Yaskawa INFORM job: R1_BATMAN_NOWY_KM-OK.JBI

/JOB
//NAME R1_BATMAN_NOWY_KM-OK
///FOLDERNAME KRIS-SCIANA
//POS
///NPOS 410,410,0,26,0,0
///TOOL 0
///POSTYPE PULSE
///PULSE
C00000=29960,139157,41546,-12188,94395,86333
C00001=12800,76505,-14321,-12731,99531,83391
C00002=-93330,-9337,26195,-7488,46800,71866
C00003=-109648,13515,16388,-582,84053,65182
C00004=-109670,16422,24252,-586,80707,65189
C00005=-109670,16934,25656,-587,80107,65191
C00006=-109670,16422,24252,-586,80707,65189
C00007=-110374,15664,24172,-576,80363,64950
C00008=-110374,13408,17598,-573,83249,64937
C00009=-100947,5020,18268,-732,78517,68109
C00010=-100947,5466,19407,-733,78046,68110
C00011=-100947,5020,18268,-732,78517,68109
C00012=-101669,3533,17505,-722,78217,67864
C00013=-100947,5020,18268,-732,78517,68109
C00014=-93324,28905,32784,-832,81932,70679
C00015=-94152,26793,37960,-831,77656,70427
C00016=-94152,27168,38874,-831,77287,70429
C00017=-94152,26793,37960,-831,77656,70427
C00018=-94428,25011,36465,-827,77656,70332
C00019=-94152,26793,37960,-831,77656,70427
C00020=-83677,18451,34531,-972,75597,74005
C00021=-83677,18852,35456,-973,75233,74007
C00022=-83677,18451,34531,-972,75597,74005
C00023=-84064,17163,33488,-967,75571,73871
C00024=-83677,18451,34531,-972,75597,74005
C00025=-81641,11244,27675,-995,76137,74695
C00026=-81493,11059,28179,-998,75733,74748
C00027=-81641,11244,27675,-995,76137,74695
C00028=-82191,12588,29665,-991,75598,74510
C00029=-81641,11244,27675,-995,76137,74695
C00030=-91711,-19484,9455,-889,71442,71303
C00031=-91372,-20164,10041,-896,70736,71423
C00032=-91711,-19484,9455,-889,71442,71303
C00033=-92389,-17223,12578,-883,70676,71076
C00034=-91711,-19484,9455,-889,71442,71303
C00035=-106821,23381,33578,-700,78719,66116
C00036=-140607,-14296,8355,17640,72856,-28938
C00037=-138803,-8748,20112,18029,68291,-28986
C00038=-139069,-9638,20936,18155,67425,-29218
C00039=-138803,-8748,20112,18029,68291,-28986
C00040=-138658,-6539,23170,18113,67548,-29051
C00041=-138803,-8748,20112,18029,68291,-28986
C00042=-151062,6621,28732,17951,73370,-32606
C00043=-147529,16835,48440,18711,66071,-32499
C00044=-147718,16293,48665,18768,65717,-32627
C00045=-147529,16835,48440,18711,66071,-32499
C00046=-147292,19253,51437,18794,65449,-32517
C00047=-147529,16835,48440,18711,66071,-32499
C00048=-160315,9548,45137,18676,67160,-36871
C00049=-160315,11416,48596,18832,66051,-37055
C00050=-160034,10639,48797,18917,65496,-37052
C00051=-160315,11416,48596,18832,66051,-37055
C00052=-159902,14249,52211,18957,65234,-37046
C00053=-160315,11416,48596,18832,66051,-37055
C00054=-160315,1266,28928,18053,72602,-36008
C00055=-155372,33863,69589,13242,72639,-71520
C00056=-155372,33877,69614,13243,72631,-71521
C00057=-155632,33114,69495,13228,72357,-71637
C00058=-155372,33877,69614,13243,72631,-71521
C00059=-154967,38534,75787,13400,71201,-71548
C00060=-155372,33877,69614,13243,72631,-71521
C00061=-155372,14771,31861,12741,85721,-70138
C00062=-144854,-16074,11616,14078,80727,-67113
C00063=-144738,-11911,19372,14194,78150,-67371
C00064=-144388,-8955,22802,14262,77515,-67327
C00065=-144738,-11911,19372,14194,78150,-67371
C00066=-145031,-12965,19294,14184,77720,-67519
C00067=-144738,-11911,19372,14194,78150,-67371
C00068=-144738,-22241,-3507,13967,86670,-66398
C00069=-137755,-5473,21324,14836,78997,-64910
C00070=-137072,-7723,19533,14904,78825,-64700
C00071=-137755,-5473,21324,14836,78997,-64910
C00072=-137755,-4185,24016,14880,78032,-65028
C00073=-137755,-5473,21324,14836,78997,-64910
C00074=-136397,694,15927,14772,85041,-63716
C00075=-136397,302,14935,14766,85437,-63669
C00076=-109887,-1557,13389,16194,80395,55204
C00077=-88793,-1230,14928,-10868,86441,64286
C00078=-87997,13509,39457,-13767,84419,65011
C00079=-88765,12150,38219,-13907,84356,64763
C00080=-87997,13509,39457,-13767,84419,65011
C00081=-87997,14649,41772,-13784,83604,65104
C00082=-87997,13509,39457,-13767,84419,65011
C00083=-87997,4090,18260,-13774,92399,64126
C00084=-90135,-15090,27302,-19288,66922,75027
C00085=-93339,-8581,40987,-20291,61446,74887
C00086=-93414,13551,61682,-18148,70133,73308
C00087=-93501,10236,57492,-18075,70950,73153
C00088=-74509,-9574,47474,-19286,61435,81215
C00089=-71490,563,57958,-19102,60836,82318
C00090=-73930,26348,84328,-20021,57559,82128
C00091=-53296,23546,81196,-16554,61634,87978
C00092=-53399,1993,45500,-15348,72112,86487
C00093=-93772,6441,51176,-23543,71504,29074
C00094=-93782,7493,53021,-23621,70954,29184
C00095=-97809,11823,34750,-18310,96930,22381
C00096=-97765,18036,47284,-18125,92636,23039
C00097=-93436,10227,57510,-23741,69792,29543
C00098=-92885,10092,58329,-23719,69400,29810
C00099=-94577,32380,63989,-17035,90534,24406
C00100=-93990,31397,63393,-16840,90513,24603
C00101=-86403,12665,47397,-14267,92055,26863
C00102=-83940,7836,43519,-13404,92349,27621
C00103=-88022,26657,64193,-8590,95838,24607
C00104=-86621,7360,57775,-7913,90052,25407
C00105=-86874,-9205,28605,-8179,99382,24730
C00106=-93784,11972,60674,-23958,68741,29649
C00107=-120720,1752,25513,-527,80353,-9094
C00108=-141476,7352,24714,17219,80156,-38332
C00109=-140652,10872,31760,17392,77568,-38413
C00110=-151911,2048,28558,16772,77396,-42350
C00111=-153373,1194,28316,16661,77408,-42852
C00112=-154278,885,28252,16586,77468,-43151
C00113=-151033,405,27146,8511,73769,-41301
C00114=-151062,615,27322,8509,73772,-41310
C00115=-152803,25350,52147,11197,72163,-42431
C00116=-157202,33761,63402,16632,73491,-44702
C00117=-172575,32003,68245,15007,72491,-49961
C00118=-172661,17404,41016,14506,81470,-48897
C00119=-145328,-17018,3942,17006,81208,-68726
C00120=-143820,-16511,8308,17205,78576,-68574
C00121=-147802,-4731,19998,17005,78294,-69996
C00122=-143624,-15596,9649,11345,73102,-68510
C00123=-152471,-38163,-4132,7931,70088,-70764
C00124=-152752,-37985,-4023,7933,70138,-70858
C00125=-161611,-21890,10565,15904,78087,-74768
C00126=-170415,38593,75058,15377,71350,-78588
C00127=-170289,22176,44233,14795,81516,-77278
C00128=-170289,11960,19922,14705,90922,-76157
C00129=16919,130033,39084,-10517,94456,75601
C00130=16919,130033,39084,-10517,94456,75601
C00131=-97369,-13902,24194,28978,70576,-6709
C00132=-95632,-2500,42487,30176,65295,-7505
C00133=-95207,2788,47639,30323,64767,-7497
C00134=-94456,3304,48081,30401,64521,-7286
C00135=-95207,2788,47639,30323,64767,-7497
C00136=-94939,4605,50640,30565,63888,-7653
C00137=-95207,2788,47639,30323,64767,-7497
C00138=-103162,11339,55190,29411,67038,-9800
C00139=-102527,20996,70482,30499,62962,-10725
C00140=-102527,23747,75000,30853,61778,-11081
C00141=-102527,20996,70482,30499,62962,-10725
C00142=-101170,23554,74068,30934,61779,-10587
C00143=-102527,20996,70482,30499,62962,-10725
C00144=-108080,-3135,57545,30673,60740,-13355
C00145=-107519,-2528,59016,30963,60068,-13361
C00146=-108080,-3135,57545,30673,60740,-13355
C00147=-108548,-1030,60547,30798,60211,-13680
C00148=-108080,-3135,57545,30673,60740,-13355
C00149=-118454,-19329,55183,30459,57655,-17824
C00150=-117324,-18814,56509,30922,56888,-17699
C00151=-118454,-19329,55183,30459,57655,-17824
C00152=-118779,-17072,58124,30582,57172,-18080
C00153=-118454,-19329,55183,30459,57655,-17824
C00154=-119568,-37031,32608,28877,62130,-16877
C00155=-139069,-33471,54850,26577,56126,-24455
C00156=-140948,-25344,66415,26849,53845,-25589
C00157=-140947,-22345,70767,27227,52824,-25875
C00158=-140948,-25344,66415,26849,53845,-25589
C00159=-138778,-24772,68372,27918,52625,-25364
C00160=-140948,-28933,61200,26421,55072,-25252
C00161=-139172,-36190,52504,26531,56189,-82791
C00162=-107699,-48855,44139,22027,38536,-72276
C00163=-109632,-48276,45968,22227,38076,-73074
C00164=-107699,-48855,44139,22027,38536,-72276
C00165=-107022,-47413,45796,22221,38170,-72148
C00166=-107699,-48855,44139,22027,38536,-72276
C00167=-87180,-57379,25744,20107,41611,-64125
C00168=-87177,-56321,27969,20431,40831,-64319
C00169=-87180,-57379,25744,20107,41611,-64125
C00170=-86636,-54726,28428,20224,41246,-64016
C00171=-87180,-57379,25744,20107,41611,-64125
C00172=-68556,-59148,10398,16762,46593,-56068
C00173=-68720,-58452,12286,16994,45847,-56271
C00174=-68556,-59148,10398,16762,46593,-56068
C00175=-67991,-57295,12403,16799,46232,-55922
C00176=-68556,-59148,10398,16762,46593,-56068
C00177=-65065,-64227,-6791,14726,53714,-53588
C00178=-61076,-57425,2885,14865,50705,-52539
C00179=-61164,-57495,4364,15074,49802,-52712
C00180=-61076,-57425,2885,14865,50705,-52539
C00181=-60686,-55325,4818,14851,50535,-52416
C00182=-61076,-57425,2885,14865,50705,-52539
C00183=-61076,-73603,-22996,13552,58097,-51511
C00184=-82396,-73217,-22842,14872,61637,60164
C00185=-87516,-60977,-6284,80955,41162,78434
C00186=-74092,-52490,8277,91201,32262,75613
C00187=-78785,-42356,17001,89628,35140,75415
C00188=-77330,-41476,17474,89941,34254,75571
C00189=-78785,-42356,17001,89628,35140,75415
C00190=-78785,-39715,21246,91443,35108,74420
C00191=-78785,-42356,17001,89628,35140,75415
C00192=-88814,-14584,37421,84097,41483,76258
C00193=-87600,-13774,38015,84402,40735,76362
C00194=-88814,-14584,37421,84097,41483,76258
C00195=-88814,-11485,42642,85948,41288,75148
C00196=-88814,-14584,37421,84097,41483,76258
C00197=-88814,-12912,40245,85098,41370,75657
C00198=-87720,-12181,40790,85402,40703,75739
C00199=-88814,-12912,40245,85098,41370,75657
C00200=-88814,-10194,44789,86704,41222,74694
C00201=-88814,-12912,40245,85098,41370,75657
C00202=-81268,8239,25602,62836,54247,42871
C00203=-99383,-12682,5103,58765,66557,41036
C00204=-74635,2773,19953,61588,50422,44547
C00205=-74870,7103,29898,71541,48579,40569
C00206=-73722,4389,21160,61383,49897,44786
C00207=-73275,4966,21408,61205,49691,44957
C00208=-83489,55985,81914,76438,52196,35596
C00209=-80400,36125,52423,64197,52680,41941
C00210=-80398,36126,52424,64197,52679,41941
C00211=-78951,-40444,4950,38310,62421,-17800
C00212=-78960,-34903,14668,39360,59955,-18811
C00213=-72845,-10333,24086,24565,76568,-49529
C00214=-69730,1194,40732,25450,71769,-49472
C00215=-79919,-36306,13442,39288,60368,-19058
C00216=-79943,-36084,12678,39084,60835,-18874
C00217=-86153,35123,85647,24141,66737,-56179
C00218=-71006,-12268,19845,19209,73235,-48605
C00219=-78486,-5699,27880,17849,72527,-51167
C00220=-84137,3114,38840,17597,71558,-53260
C00221=-84122,-12372,4412,16852,84221,-51450
C00222=-94700,16963,33528,63705,62536,40249
C00223=-80389,36149,52448,64198,52673,41941
C00224=-80398,36126,52424,64197,52679,41941
C00225=-82543,39244,62629,76344,52787,36963
C00226=-83474,48309,76175,82007,53048,34101
C00227=-80829,34452,49584,63632,53361,42311
C00228=-80419,35008,49905,63542,53144,42433
C00229=-83495,46424,73588,81542,53170,34449
C00230=-83461,45298,72093,81297,53209,34643
C00231=-83534,45148,71928,81265,53263,34652
C00232=-83974,39234,63618,79687,53967,35775
C00233=-87946,20987,32632,62140,59518,42667
C00234=-98278,19923,28034,11913,78019,-9874
C00235=-92244,58536,75756,7832,70371,-3504
C00236=-91977,78904,104422,8238,63238,-3903
C00237=-107781,18098,54792,50122,40570,-59241
C00238=-108140,20187,57804,50894,40242,-59767
C00239=-92594,57126,80356,8020,66880,-3859
C00240=-94908,21990,48768,7976,68471,-4548
C00241=-98306,-6406,30616,8206,65402,-5929
C00242=-103070,-28468,23138,8725,59186,-8038
C00243=-105710,-35465,21971,8985,56591,-9160
C00244=-105525,-39817,14322,8753,59014,-8895
C00245=-105525,-70728,-42035,7727,77630,-7598
C00246=-78386,25843,42020,64423,60972,44329
C00247=-85759,14880,31595,64053,66010,43452
C00248=-85595,16938,42729,82497,65241,37214
C00249=-81136,28617,59931,85714,61589,35095
C00250=-78173,23730,38609,63927,61301,44837
C00251=-78597,23175,38323,63988,61519,44714
C00252=-72881,-4192,29043,86400,56225,36548
C00253=-67760,-16410,19348,87784,52710,36541
C00254=-59662,-27119,-2583,63857,48640,46851
C00255=-59488,-28058,-2749,64137,48352,46679
C00256=-60158,-29069,10200,71536,45362,41690
C00257=-61387,-28761,11042,71804,46022,41293
C00258=-67092,-34207,-766,67938,51323,42934
C00259=-57818,-28976,-3296,38246,61056,30495
C00260=-70399,-33004,-19929,37727,73042,29338
C00261=-119023,5793,43031,54634,61324,54134
C00262=-110425,23913,49460,37198,87531,-1667
C00263=-103784,36935,71027,39124,79569,-1855
C00264=-107895,22032,60540,56797,53926,55382
C00265=-107775,18111,54805,55911,54728,56108
C00266=-104144,33311,68301,39058,79572,-1995
C00267=-105177,26013,62623,38825,79784,-2330
C00268=-105381,26208,63001,38785,79763,-2415
C00269=-106285,20699,59223,38608,79730,-2777
C00270=-106624,19858,58731,38534,79764,-2897
C00271=-106746,20912,59987,38524,79628,-2990
C00272=-106325,7794,45978,38293,75046,-4276
C00273=-104338,-11348,28641,37974,64498,-6611
C00274=-104860,-11037,29608,38068,64365,-6884
C00275=-107519,-11058,32205,38335,64151,-8093
C00276=-107851,-11129,32812,38426,63958,-8307
C00277=-116434,-38739,5593,36913,69412,-9812
C00278=-124683,-63657,-10921,36340,70465,-12735
C00279=-150183,-86751,-58871,11994,78291,3293
C00280=-2356,-86751,-58871,11994,78291,3293
C00281=12334,49205,1562,-2559,87983,53268
C00282=-150183,-86751,-58871,11994,78291,3293
C00283=-131366,13830,22994,-19726,75607,38471
C00284=-136534,55496,89709,-36696,55641,43467
C00285=-137035,56054,90375,-36738,55351,43362
C00286=-136534,55496,89709,-36696,55641,43467
C00287=-136534,59618,96436,-37542,54010,44136
C00288=-136534,55496,89709,-36696,55641,43467
C00289=-145752,56924,83291,-5552,58900,12813
C00290=-147360,56365,85008,-5446,57459,12300
C00291=-147195,60965,91580,-5568,55798,12447
C00292=-147360,56365,85008,-5446,57459,12300
C00293=-147752,57421,87154,-5449,56660,12196
C00294=-147360,56365,85008,-5446,57459,12300
C00295=-144876,20699,52980,-5661,58991,13126
C00296=-144465,22925,56598,-5771,57941,13331
C00297=-144876,20699,52980,-5661,58991,13126
C00298=-145346,20760,54373,-5658,58141,13001
C00299=-144876,20699,52980,-5661,58991,13126
C00300=-140458,-9363,35089,-6525,54898,15024
C00301=-139844,-7295,37930,-6647,54260,15291
C00302=-140458,-9363,35089,-6525,54898,15024
C00303=-141162,-9224,36313,-6501,54169,14811
C00304=-140458,-9363,35089,-6525,54898,15024
C00305=-124022,-11653,42832,-20763,58582,23587
C00306=-123999,-9443,45795,-20909,57941,23722
C00307=-124022,-11653,42832,-20763,58582,23587
C00308=-124750,-10986,44233,-20923,57940,23461
C00309=-124022,-11653,42832,-20763,58582,23587
C00310=-120425,-27436,23026,-19779,63062,73790
C00311=-124426,-21462,36323,-21031,57405,73472
C00312=-124464,-21490,37251,-21166,56849,73573
C00313=-124426,-21462,36323,-21031,57405,73472
C00314=-125014,-20092,38108,-21159,56911,73366
C00315=-124426,-21462,36323,-21031,57405,73472
C00316=-142818,-53721,4956,-21021,55965,67145
C00317=-142626,-53506,6347,-21202,55310,67354
C00318=-142818,-53721,4956,-21021,55965,67145
C00319=-143779,-52181,6747,-21095,55463,66895
C00320=-142818,-53721,4956,-21021,55965,67145
C00321=-174971,-75680,-15206,-18859,50174,56027
C00322=-175130,-75408,-13794,-19036,49449,56108
C00323=-174971,-75680,-15206,-18859,50174,56027
C00324=-175277,-74010,-13504,-18872,49932,55952
C00325=-174971,-75680,-15206,-18859,50174,56027
C00326=-173245,-86721,-27893,-18523,52547,56249
C00327=-203888,-83968,-26454,-13077,47682,44754
C00328=-205019,-83483,-25221,-12917,47022,44380
C00329=-203888,-83968,-26454,-13077,47682,44754
C00330=-204234,-82255,-25110,-12985,47684,44611
C00331=-203888,-83968,-26454,-13077,47682,44754
C00332=-178857,-84729,-36876,-16471,57715,53184
C00333=-172192,-78951,-17187,-49367,43626,66497
C00334=-173896,-78013,-16876,-49026,43021,65876
C00335=-172192,-78951,-17187,-49367,43626,66497
C00336=-172192,-77329,-14763,-49894,43190,66824
C00337=-172192,-78951,-17187,-49367,43626,66497
C00338=-162487,-85150,-21286,-50022,47755,69383
C00339=-141360,-58545,-9704,-51911,39719,82506
C00340=-155475,-48260,1081,-49396,31731,78582
C00341=-156810,-47533,1467,-48693,31169,77981
C00342=-155475,-48260,1081,-49396,31731,78582
C00343=-155475,-46586,3939,-50523,31140,79172
C00344=-155475,-48260,1081,-49396,31731,78582
C00345=-143506,-57069,-7972,-51767,38422,82026
C00346=-132998,-15066,34811,-73278,45446,90463
C00347=-136647,7793,53326,-73557,43352,89771
C00348=-137414,8138,53635,-73690,42883,89678
C00349=-136647,7793,53326,-73557,43352,89771
C00350=-136647,9971,57074,-74779,42995,90526
C00351=-136647,7793,53326,-73557,43352,89771
C00352=-127315,-7809,27658,-65953,51971,86730
C00353=-123754,-52231,-17316,-40750,89865,-5838
C00354=-130215,-25533,26580,-55595,80666,-780
C00355=-127399,30151,75869,-54823,81081,357
C00356=-123761,23089,64182,-53294,85068,-318
C00357=-107579,-13362,25214,-39024,97613,11163
C00358=-170043,-71406,-31414,-11284,81739,48155
C00359=-190061,-61831,-15348,-14174,73926,42337
C00360=-162764,-46045,3348,-10421,74427,51168
C00361=-141001,-25000,21572,-6477,76090,57905
C00362=-128005,1092,47071,-3936,74564,61986
C00363=-123328,16053,63213,-3007,72497,63466
C00364=-123444,-5699,22378,-2915,86428,63100
C00365=-123444,-16678,-3411,-2947,96644,62863
C00366=-133517,-66572,-32265,-38878,44642,78881
C00367=-132900,-49128,-445,-67646,40881,87931
C00368=-134943,-41043,7919,-68788,39256,88202
C00369=-129486,24309,60482,-67313,43043,88408
C00370=-129295,28550,64902,-67843,42938,88773
C00371=-124005,7439,40047,-63776,48062,87191
C00372=-119115,-2939,24898,-61013,52949,86096
C00373=-132234,15475,18840,-9177,73687,21564
C00374=-138193,54177,73040,-9110,59720,20493
C00375=-142429,56695,78528,-2248,54886,15330
C00376=-135428,11470,41007,-7421,55168,18590
C00377=-124358,-15323,27893,-15893,51961,24324
C00378=-114489,-24173,28344,-21843,50628,29378
C00379=-104693,-29158,30498,-25923,50747,33967
C00380=-104394,-36428,19495,-24933,53579,33323
C00381=-104394,-63765,-28743,-21562,68022,30158
C00382=-137801,-54017,-22800,-32811,77180,42551
C00383=-145098,-49977,-15343,-33510,72300,41124
C00384=-157536,-82053,-30611,-35478,61676,39542
C00385=-167332,-94403,-34954,-36782,54951,37849
C00386=-168775,-95552,-35063,-36976,53981,37598
C00387=-175265,-101786,-36159,-35767,45251,37123
C00388=-172094,-106020,-33228,-38547,43201,39696
C00389=-170782,-105999,-32632,-38876,43404,40255
C00390=-154100,-109404,-39309,-37897,51447,44344
C00391=-127200,-116118,-56301,-33842,67042,49701
C00392=-160521,-112920,-64126,-13181,65496,7682
C00393=-193283,-91966,-46197,-10210,60672,-3708
C00394=-179428,-87326,-33956,-22991,51575,4568
C00395=-182309,-93219,-32914,-23693,47463,4374
C00396=-181968,-93619,-32743,-23870,47264,4575
C00397=-184128,-96951,-32374,-24207,44941,4267
C00398=-184601,-97825,-32091,-24365,44249,4253
C00399=-192271,-94092,-34086,-15205,49403,-1377
C00400=-156461,-94996,-22149,-46235,47288,20425
C00401=-143339,-75495,-15964,-42086,57329,21373
C00402=-155681,-87382,-19579,-43513,38484,12104
C00403=-154383,-87178,-18470,-44197,38599,12813
C00404=-148677,-87335,-15888,-46202,39785,15423
C00405=-143679,-101658,-25353,-47688,40824,17641
C00406=-91918,-122697,-50228,-39868,65277,29334
C00407=-93784,-22748,-9129,-22507,91967,25137
C00408=5840,107598,31668,-14199,93922,74405
C00409=29960,139157,41546,-12188,94395,86333
BC00000=68533,13783,1075157
BC00001=137001,15545,1050957
BC00002=200108,21911,920879
BC00003=200107,21911,776849
BC00004=200107,21911,776849
BC00005=200107,21911,776849
BC00006=200107,21911,776849
BC00007=200107,21911,776849
BC00008=200107,21911,776849
BC00009=199824,21894,777489
BC00010=199824,21894,777489
BC00011=199824,21894,777489
BC00012=199824,21894,777489
BC00013=199824,21894,777489
BC00014=199824,21894,743092
BC00015=199824,21894,743092
BC00016=199824,21894,743092
BC00017=199824,21894,743092
BC00018=199824,21894,743092
BC00019=199824,21894,743092
BC00020=199824,21894,743092
BC00021=199824,21894,743092
BC00022=199824,21894,743092
BC00023=199824,21894,743092
BC00024=199824,21894,743092
BC00025=199824,21894,743092
BC00026=199824,21894,743092
BC00027=199824,21894,743092
BC00028=199824,21894,743092
BC00029=199824,21894,743092
BC00030=199824,21894,835261
BC00031=199824,21894,835261
BC00032=199824,21894,835261
BC00033=199824,21894,835261
BC00034=199824,21894,835261
BC00035=199824,21894,835261
BC00036=199824,21894,835261
BC00037=199824,21894,835261
BC00038=199824,21894,835261
BC00039=199824,21894,835261
BC00040=199824,21894,835261
BC00041=199824,21894,835261
BC00042=199824,21894,835261
BC00043=199824,21894,835261
BC00044=199824,21894,835261
BC00045=199824,21894,835261
BC00046=199824,21894,835261
BC00047=199824,21894,835261
BC00048=199824,21894,835261
BC00049=199824,21894,835261
BC00050=199824,21894,835261
BC00051=199824,21894,835261
BC00052=199824,21894,835261
BC00053=199824,21894,835261
BC00054=199824,21894,835261
BC00055=199824,21894,835261
BC00056=199824,21894,835261
BC00057=199824,21894,835261
BC00058=199824,21894,835261
BC00059=199824,21894,835261
BC00060=199824,21894,835261
BC00061=199824,21894,835261
BC00062=199824,21894,835261
BC00063=199824,21894,835261
BC00064=199824,21894,835261
BC00065=199824,21894,835261
BC00066=199824,21894,835261
BC00067=199824,21894,835261
BC00068=199824,21894,835261
BC00069=199824,21895,835258
BC00070=199824,21895,835258
BC00071=199824,21895,835258
BC00072=199824,21895,835258
BC00073=199824,21895,835258
BC00074=199824,21895,835258
BC00075=199824,21895,835258
BC00076=199824,21895,835258
BC00077=199824,21895,835258
BC00078=199824,21895,835258
BC00079=199824,21895,835258
BC00080=199824,21895,835258
BC00081=199824,21895,835258
BC00082=199824,21895,835258
BC00083=199824,21895,835258
BC00084=205692,85135,967220
BC00085=205692,85135,967220
BC00086=205692,85135,967220
BC00087=205692,85135,967220
BC00088=205902,84947,966975
BC00089=205902,84947,966975
BC00090=205902,84947,966975
BC00091=205901,84948,926900
BC00092=205901,84948,926900
BC00093=218485,27554,1075175
BC00094=218485,27554,989857
BC00095=212076,30602,851577
BC00096=212076,30602,851577
BC00097=212075,30604,960971
BC00098=212075,30604,960971
BC00099=212076,30603,851574
BC00100=212076,30603,851574
BC00101=212076,30603,851572
BC00102=212076,30603,851571
BC00103=212076,30603,851571
BC00104=269506,91403,851571
BC00105=269506,91403,851571
BC00106=228143,33934,978152
BC00107=228143,33934,890863
BC00108=228143,33934,823600
BC00109=228143,33934,823600
BC00110=228143,33934,823600
BC00111=228143,33934,823600
BC00112=228143,33934,823600
BC00113=228143,33934,823600
BC00114=228143,33934,823600
BC00115=228144,33934,823598
BC00116=228144,33934,823598
BC00117=228144,33934,823598
BC00118=228144,33934,823598
BC00119=228144,33934,823598
BC00120=228144,33934,823598
BC00121=228144,33934,823598
BC00122=228144,33934,823598
BC00123=228144,33934,823598
BC00124=228144,33934,823598
BC00125=228144,33934,823598
BC00126=228144,33934,823598
BC00127=228144,33934,823598
BC00128=228144,33934,918948
BC00129=81693,35088,1064811
BC00130=81693,35088,1064811
BC00131=268670,144197,1015710
BC00132=268670,144197,1015710
BC00133=268670,144197,1015710
BC00134=268670,144197,1015710
BC00135=268670,144197,1015710
BC00136=268670,144197,1015710
BC00137=268670,144197,1015710
BC00138=268670,144196,1015709
BC00139=268670,144196,1015709
BC00140=268670,144196,1015709
BC00141=268670,144196,1015709
BC00142=268670,144196,1015709
BC00143=268670,144196,1015709
BC00144=268670,144196,1015709
BC00145=268669,144195,1015708
BC00146=268670,144196,1015709
BC00147=268670,144196,1015709
BC00148=268670,144196,1015709
BC00149=268670,144196,1015709
BC00150=268670,144196,1015709
BC00151=268670,144196,1015709
BC00152=268670,144196,1015709
BC00153=268670,144196,1015709
BC00154=268670,144196,1015709
BC00155=268670,144196,1015709
BC00156=268670,144196,1015709
BC00157=268670,144196,1015708
BC00158=268670,144196,1015709
BC00159=268670,144196,1015709
BC00160=268670,144196,1015709
BC00161=268670,144196,1015709
BC00162=268670,144196,1015709
BC00163=268670,144196,1015709
BC00164=268670,144196,1015709
BC00165=268670,144196,1015709
BC00166=268670,144196,1015709
BC00167=268669,113243,1015707
BC00168=268669,113243,1015707
BC00169=268669,113243,1015707
BC00170=268669,113243,1015707
BC00171=268669,113243,1015707
BC00172=268670,72970,1015708
BC00173=268670,72970,1015708
BC00174=268670,72970,1015708
BC00175=268670,72970,1015708
BC00176=268670,72970,1015708
BC00177=268670,48316,1015709
BC00178=268670,48316,1015709
BC00179=268670,48316,1015709
BC00180=268670,48316,1015709
BC00181=268670,48316,1015709
BC00182=268670,48316,1015709
BC00183=268670,48316,1015709
BC00184=268670,48316,1015709
BC00185=220078,15,922795
BC00186=227337,15,912089
BC00187=230240,15,907806
BC00188=230240,15,907806
BC00189=230240,15,907806
BC00190=230240,15,907806
BC00191=230240,15,907806
BC00192=230240,50273,907806
BC00193=230240,50273,907806
BC00194=230240,50273,907806
BC00195=230240,50273,907806
BC00196=230240,50273,907806
BC00197=230240,113905,907806
BC00198=230240,113905,907806
BC00199=230240,113905,907806
BC00200=230240,113905,907806
BC00201=230240,113905,907806
BC00202=173944,15,921053
BC00203=173944,15,921053
BC00204=178824,15,792329
BC00205=180775,15,783854
BC00206=180775,15,783854
BC00207=180775,15,783854
BC00208=180775,20545,783854
BC00209=179033,31181,784483
BC00210=174154,30731,805671
BC00211=235405,15,1075175
BC00212=235405,15,1001205
BC00213=235405,15,1001205
BC00214=235405,15,1001205
BC00215=243821,15,976624
BC00216=243821,15,976624
BC00217=235405,15,1001205
BC00218=196817,56536,842735
BC00219=189615,67087,813156
BC00220=189615,67087,813156
BC00221=189615,67087,813156
BC00222=174140,26317,913732
BC00223=174140,26317,913732
BC00224=174140,26317,806198
BC00225=179019,26768,785009
BC00226=180971,26948,776534
BC00227=180971,26948,776534
BC00228=180971,26948,776534
BC00229=181150,62034,771629
BC00230=181286,88704,767900
BC00231=181286,91968,766556
BC00232=177104,86088,775373
BC00233=174349,92139,798351
BC00234=257727,78000,903004
BC00235=258272,77360,890255
BC00236=258272,77360,890255
BC00237=262417,85815,884854
BC00238=262417,85815,884854
BC00239=258272,77360,890254
BC00240=258271,77360,890253
BC00241=258271,77360,890253
BC00242=258271,77360,890253
BC00243=258271,77360,890253
BC00244=258271,77360,890253
BC00245=258271,77360,890253
BC00246=174013,15,918199
BC00247=174013,15,810664
BC00248=180838,15,781222
BC00249=180838,15,781222
BC00250=180838,15,781222
BC00251=180838,15,781222
BC00252=180838,15,781222
BC00253=180838,15,781222
BC00254=180838,15,781222
BC00255=180838,15,781222
BC00256=180838,15,836511
BC00257=180838,15,836511
BC00258=180838,15,836511
BC00259=197117,15,902644
BC00260=197118,16,902641
BC00261=268113,94143,1075175
BC00262=276934,120699,948945
BC00263=276934,120699,948945
BC00264=274036,93127,945393
BC00265=274036,93127,945393
BC00266=276934,120699,948945
BC00267=276934,120699,948945
BC00268=276934,120699,948945
BC00269=276934,120699,948945
BC00270=276934,120699,948945
BC00271=276934,120699,948945
BC00272=276967,133711,947374
BC00273=277023,156083,944672
BC00274=277023,156083,944672
BC00275=277023,156083,944672
BC00276=277023,156083,944672
BC00277=277023,156083,944672
BC00278=277023,156083,944672
BC00279=277023,156083,944672
BC00280=135439,156083,1063650
BC00281=51795,156431,1068049
BC00282=277023,156083,944672
BC00283=173944,70115,921053
BC00284=173945,70115,925166
BC00285=173945,70115,925166
BC00286=173945,70115,925166
BC00287=173945,70115,925166
BC00288=173945,70115,925166
BC00289=173945,70115,921050
BC00290=173945,70115,921050
BC00291=173945,70115,921050
BC00292=173945,70115,921050
BC00293=173945,70115,921050
BC00294=173945,70115,921050
BC00295=173945,70115,921050
BC00296=173945,70115,921050
BC00297=173945,70115,921050
BC00298=173945,70115,921050
BC00299=173945,70115,921050
BC00300=173945,70115,921050
BC00301=173945,70115,921050
BC00302=173945,70115,921050
BC00303=173945,70115,921050
BC00304=173945,70115,921050
BC00305=173945,70115,921050
BC00306=173945,70115,921050
BC00307=173945,70115,921050
BC00308=173945,70115,921050
BC00309=173945,70115,921050
BC00310=173945,70115,921050
BC00311=173945,70115,921050
BC00312=173945,70115,921050
BC00313=173945,70115,921050
BC00314=173945,70115,921050
BC00315=173945,70115,921050
BC00316=173945,70115,921050
BC00317=173945,70115,921050
BC00318=173945,70115,921050
BC00319=173945,70115,921050
BC00320=173945,70115,921050
BC00321=173945,70115,921050
BC00322=173945,70115,921050
BC00323=173945,70115,921050
BC00324=173945,70115,921050
BC00325=173945,70115,921050
BC00326=173945,70115,921050
BC00327=173946,70115,921047
BC00328=173946,70115,921047
BC00329=173946,70115,921047
BC00330=173946,70115,921047
BC00331=173946,70115,921047
BC00332=173945,70114,921040
BC00333=173945,70114,921040
BC00334=173945,70114,921040
BC00335=173945,70114,921040
BC00336=173945,70114,921040
BC00337=173945,70114,921040
BC00338=173945,70114,921040
BC00339=173945,70114,921040
BC00340=173945,70114,921040
BC00341=173945,70114,921040
BC00342=173945,70114,921040
BC00343=173945,70114,921040
BC00344=173945,70114,921040
BC00345=173945,70114,921040
BC00346=173945,70114,921040
BC00347=173945,70114,921040
BC00348=173945,70114,921040
BC00349=173945,70114,921040
BC00350=173945,70114,921040
BC00351=173945,70114,921040
BC00352=173945,70114,921040
BC00353=153115,57298,944672
BC00354=153115,57298,944672
BC00355=153115,57298,944672
BC00356=153115,57298,944672
BC00357=153115,57298,944672
BC00358=153115,57298,944672
BC00359=153116,57298,944671
BC00360=153116,57298,944671
BC00361=153116,57298,916437
BC00362=153116,57298,892257
BC00363=153116,57298,881120
BC00364=153116,57298,881120
BC00365=153116,57298,881120
BC00366=153116,57298,881120
BC00367=153116,57298,881120
BC00368=153116,57298,881120
BC00369=153116,57298,881120
BC00370=153116,57298,881120
BC00371=153116,57298,881120
BC00372=153116,57298,881120
BC00373=153116,57298,881120
BC00374=153116,57298,881120
BC00375=153116,57298,881120
BC00376=153116,57299,881116
BC00377=153116,57299,881118
BC00378=153116,57298,881119
BC00379=153116,57298,881120
BC00380=153116,57298,881120
BC00381=153116,57298,881120
BC00382=153116,57298,881120
BC00383=153116,57298,881120
BC00384=153116,57298,881120
BC00385=153116,57298,881120
BC00386=153116,57298,881120
BC00387=153116,57298,881120
BC00388=153116,57298,881120
BC00389=153116,57298,881120
BC00390=153116,57298,881120
BC00391=153116,57298,881120
BC00392=155122,228922,881120
BC00393=155122,228922,881120
BC00394=155122,228922,881120
BC00395=155122,228922,881120
BC00396=155122,228922,881120
BC00397=155122,228922,881120
BC00398=155122,228922,881120
BC00399=155122,228922,881120
BC00400=155121,228922,881118
BC00401=155121,228922,881118
BC00402=155121,228922,881118
BC00403=155121,228922,881118
BC00404=155121,228922,881118
BC00405=155121,228922,881118
BC00406=155107,227689,881118
BC00407=228143,33934,978152
BC00408=99644,17711,1056249
BC00409=68533,13783,1075157
///POSTYPE BASE
///RECTAN
///RCONF 0,0,0,0,1,0,0,0,0,0,0,0,0,0,0,0,0,0,0,0,0,0,0,0
P00006=2.006,1.622,-0.565,0.0000,0.0000,0.0000
P00021=0.073,2.058,-0.109,0.0000,0.0000,0.0000
P00022=2.006,1.622,-0.565,0.0000,0.0000,0.0000
///RCONF 0,0,0,0,0,0,0,0,0,0,0,0,0,0,0,0,0,0,0,0,0,0,0,0
P00023=-2.957,-4.083,2.762,0.0000,0.0000,0.0000
P00024=-1.466,-0.226,-0.419,0.0000,0.0000,0.0000
P00025=3.643,0.007,-2.585,0.0000,0.0000,0.0000
P00026=2.644,0.055,-2.583,0.0000,0.0000,0.0000
P00027=2.278,0.099,-4.210,0.0000,0.0000,0.0000
P00028=-1.778,-0.182,-2.050,0.0000,0.0000,0.0000
P00029=1.749,4.006,-0.261,0.0000,0.0000,0.0000
P00030=-0.014,-0.768,0.131,0.0000,0.0000,0.0000
P00031=-0.170,0.039,-0.647,0.0000,0.0000,0.0000
P00032=-0.423,0.157,3.222,0.0000,0.0000,0.0000
P00033=0.854,-1.099,3.047,0.0000,0.0000,0.0000
///RCONF 0,0,0,0,1,0,0,0,0,0,0,0,0,0,0,0,0,0,0,0,0,0,0,0
P00034=-8.151,9.743,-4.393,0.0000,0.0000,0.0000
///RCONF 0,0,0,0,0,0,0,0,0,0,0,0,0,0,0,0,0,0,0,0,0,0,0,0
P00035=0.390,-0.027,1.040,0.0000,0.0000,0.0000
P00036=-2.434,0.084,0.197,0.0000,0.0000,0.0000
P00037=-1.075,5.090,-3.949,0.0000,0.0000,0.0000
P00038=0.174,-1.527,-10.860,0.0000,0.0000,0.0000
P00039=-0.109,1.838,-0.266,0.0000,0.0000,0.0000
P00040=2.716,-0.016,3.014,0.0000,0.0000,0.0000
P00041=-0.109,0.014,0.966,0.0000,0.0000,0.0000
P00042=-0.220,0.371,-0.613,0.0000,0.0000,0.0000
P00043=-0.179,-5.890,-3.227,0.0000,0.0000,0.0000
P00044=-8.560,-7.557,-5.232,0.0000,0.0000,0.0000
P00045=-8.836,-6.632,-1.438,0.0000,0.0000,0.0000
//INST
///DATE 2023/12/14 16:11
///ATTR SC,RW
///GROUP1 RB1,BS1
NOP
'R1_BATver2(-70,-90)
'Path S1517
SFTOF
MOVJ C00000 BC00000 VJ=40.00
CALL JOB:CLEAN-R1_LONG
MOVJ C00001 BC00001 VJ=50.00
MOVJ C00002 BC00002 VJ=100.00
MOVL C00003 BC00003 V=166.7
MOVL C00004 BC00004 V=166.7
REFP 3 C00005 BC00005
CALL JOB:SEARCH-R1
SET P021 P006
SFTON P021
MOVL C00006 BC00006 V=166.7
REFP 3 C00007 BC00007
CALL JOB:SEARCH-R1
SET P021 P006
SFTON P021
MOVL C00008 BC00008 V=166.7
MOVL C00009 BC00009 V=166.7
SFTOF
'2POMIAR
REFP 3 C00010 BC00010
CALL JOB:SEARCH-R1
SET P022 P006
SFTON P022
MOVL C00011 BC00011 V=166.7
REFP 3 C00012 BC00012
CALL JOB:SEARCH-R1
SET P022 P006
SFTON P022
MOVL C00013 BC00013 V=166.7
MOVL C00014 BC00014 V=166.7
SFTOF
MOVL C00015 BC00015 V=166.7
REFP 3 C00016 BC00016
CALL JOB:SEARCH-R1
SET P024 P006
SFTON P024
MOVL C00017 BC00017 V=166.7
REFP 3 C00018 BC00018
CALL JOB:SEARCH-R1
SET P024 P006
SFTON P024
MOVL C00019 BC00019 V=166.7
MOVL C00020 BC00020 V=166.7
SFTOF
'KONIEC 3 POMIAR
REFP 3 C00021 BC00021
CALL JOB:SEARCH-R1
SET P025 P006
SFTON P025
MOVL C00022 BC00022 V=166.7
REFP 3 C00023 BC00023
CALL JOB:SEARCH-R1
SET P025 P006
SFTON P025
MOVL C00024 BC00024 V=166.7
SFTOF
MOVL C00025 BC00025 V=166.7
REFP 3 C00026 BC00026
CALL JOB:SEARCH-R1
SET P026 P006
SFTON P026
MOVL C00027 BC00027 V=166.7
REFP 3 C00028 BC00028
CALL JOB:SEARCH-R1
SET P026 P006
SFTON P026
MOVL C00029 BC00029 V=166.7
SFTOF
'POMIAR 6 P27
MOVL C00030 BC00030 V=166.7
REFP 3 C00031 BC00031
CALL JOB:SEARCH-R1
SET P027 P006
SFTON P027
MOVL C00032 BC00032 V=166.7
REFP 3 C00033 BC00033
CALL JOB:SEARCH-R1
SET P027 P006
SFTON P027
MOVL C00034 BC00034 V=166.7
MOVJ C00035 BC00035 VJ=50.00
MOVJ C00036 BC00036 VJ=50.00
MOVL C00037 BC00037 V=166.7
REFP 3 C00038 BC00038
CALL JOB:SEARCH-R1
SET P028 P006
SFTON P028
MOVL C00039 BC00039 V=166.7
REFP 3 C00040 BC00040
CALL JOB:SEARCH-R1
SET P028 P006
SFTON P028
MOVL C00041 BC00041 V=166.7
SFTOF
MOVJ C00042 BC00042 VJ=50.00
MOVJ C00043 BC00043 VJ=50.00
REFP 3 C00044 BC00044
CALL JOB:SEARCH-R1
SET P029 P006
SFTON P029
MOVL C00045 BC00045 V=166.7
REFP 3 C00046 BC00046
CALL JOB:SEARCH-R1
SET P029 P006
SFTON P029
MOVL C00047 BC00047 V=166.7
SFTOF
MOVJ C00048 BC00048 VJ=50.00
MOVL C00049 BC00049 V=166.7
REFP 3 C00050 BC00050
CALL JOB:SEARCH-R1
SET P030 P006
SFTON P030
MOVL C00051 BC00051 V=166.7
REFP 3 C00052 BC00052
CALL JOB:SEARCH-R1
SET P030 P006
SFTON P030
MOVL C00053 BC00053 V=166.7
SFTOF
MOVJ C00054 BC00054 VJ=50.00
MOVJ C00055 BC00055 VJ=50.00
MOVL C00056 BC00056 V=166.7
REFP 3 C00057 BC00057
CALL JOB:SEARCH-R1
SET P031 P006
SFTON P031
MOVL C00058 BC00058 V=166.7
REFP 3 C00059 BC00059
CALL JOB:SEARCH-R1
SET P031 P006
SFTON P031
MOVL C00060 BC00060 V=166.7
SFTOF
MOVJ C00061 BC00061 VJ=50.00
MOVJ C00062 BC00062 VJ=50.00
MOVL C00063 BC00063 V=166.7
REFP 3 C00064 BC00064
CALL JOB:SEARCH-R1
SET P032 P006
SFTON P032
MOVL C00065 BC00065 V=166.7
REFP 3 C00066 BC00066
CALL JOB:SEARCH-R1
SET P032 P006
SFTON P032
MOVL C00067 BC00067 V=166.7
SFTOF
MOVJ C00068 BC00068 VJ=50.00
MOVL C00069 BC00069 V=166.7
REFP 3 C00070 BC00070
CALL JOB:SEARCH-R1
SET P033 P006
SFTON P033
MOVL C00071 BC00071 V=166.7
REFP 3 C00072 BC00072
CALL JOB:SEARCH-R1
SET P033 P006
SFTON P033
MOVL C00073 BC00073 V=166.7
SFTOF
MOVL C00074 BC00074 V=166.7
MOVJ C00075 BC00075 VJ=30.00
MOVJ C00076 BC00076 VJ=30.00
MOVJ C00077 BC00077 VJ=30.00
MOVL C00078 BC00078 V=166.7
REFP 3 C00079 BC00079
CALL JOB:SEARCH-R1
SET P034 P006
SFTON P034
MOVL C00080 BC00080 V=166.7
REFP 3 C00081 BC00081
CALL JOB:SEARCH-R1
SET P034 P006
SFTON P034
MOVL C00082 BC00082 V=166.7
MOVL C00083 BC00083 V=166.7
'KONIEC SZUKANIA BATMANA
SFTOF
'SPAWANIE BATMANA
'SPAWANIE BATMANA
MOVJ C00084 BC00084 VJ=100.00
SFTON P021
MOVL C00085 BC00085 V=166.7 PL=0
REFP 1 C00086 BC00086
REFP 2 C00087 BC00087
MACRO1 MJ#(0) ARGF7
ARCON
SFTON P022
MOVL C00088 BC00088 V=10.8
MOVL C00089 BC00089 V=10.8
SFTON P024
MOVL C00090 BC00090 V=10.8
SFTON P025
MOVL C00091 BC00091 V=10.8
ARCOF
MOVJ C00092 BC00092 VJ=20.00
SFTOF
'Path W1538
SFTOF
'Path W1533
SFTOF
MOVJ C00093 BC00093 VJ=100.00
MOVJ C00094 BC00094 VJ=100.00
MOVJ C00095 BC00095 VJ=100.00
SFTON P034
MOVL C00096 BC00096 V=166.7 PL=0
REFP 1 C00097 BC00097
REFP 2 C00098 BC00098
MACRO1 MJ#(0) ARGF9
ARCON
MOVL C00099 BC00099 V=10.8
SFTON P034
MOVL C00100 BC00100 V=10.8
MOVL C00101 BC00101 V=10.8
MOVL C00102 BC00102 V=10.8
SFTON P027
MOVL C00103 BC00103 V=10.8
SFTON P026
MOVL C00104 BC00104 V=10.8
ARCOF
SFTOF
MOVL C00105 BC00105 V=400.0
MOVL C00106 BC00106 V=1000.0
'SPAWANIE BATMANA 2 POLOWA
MOVJ C00107 BC00107 VJ=25.00
MOVJ C00108 BC00108 VJ=25.00
SFTON P021
MOVL C00109 BC00109 V=166.7
ARCON
SFTON P028
MOVL C00110 BC00110 V=10.8
MOVL C00111 BC00111 V=10.8
ARCON
MOVL C00112 BC00112 V=10.8
MOVL C00113 BC00113 V=10.8
SFTON P029
MOVL C00114 BC00114 V=10.8
MOVL C00115 BC00115 V=10.8
MOVL C00116 BC00116 V=10.8
SFTON P030
MOVL C00117 BC00117 V=10.8
ARCOF
MOVJ C00118 BC00118 VJ=40.00
SFTOF
MOVJ C00119 BC00119 VJ=50.00
SFTON P033
MOVJ C00120 BC00120 VJ=30.00
ARCON
MOVL C00121 BC00121 V=10.8
MOVL C00122 BC00122 V=10.8
SFTON P033
MOVL C00123 BC00123 V=10.8
MOVL C00124 BC00124 V=10.8
SFTON P032
MOVL C00125 BC00125 V=10.8
SFTON P031
MOVL C00126 BC00126 V=10.8
ARCOF
MOVJ C00127 BC00127 VJ=25.00
SFTOF
MOVJ C00128 BC00128 VJ=40.00
'KONIEC SPAWANIA BATMANA
'POMIAR PRAWEGO BOCZKA -SEARCH
MOVJ C00129 BC00129 VJ=100.00
CALL JOB:CLEAN-R1_LONG
MOVJ C00130 BC00130 VJ=40.00
MOVJ C00131 BC00131 VJ=100.00
MOVJ C00132 BC00132 VJ=100.00
MOVL C00133 BC00133 V=60.0
REFP 3 C00134 BC00134
CALL JOB:SEARCH-R1
SET P030 P006
SFTON P030
MOVL C00135 BC00135 V=166.7
REFP 3 C00136 BC00136
CALL JOB:SEARCH-R1
SET P030 P006
SFTON P030
MOVL C00137 BC00137 V=166.7
SFTOF
'Path S1526
SFTOF
MOVL C00138 BC00138 V=166.7
MOVL C00139 BC00139 V=166.7
REFP 3 C00140 BC00140
CALL JOB:SEARCH-R1
SET P031 P006
SFTON P031
MOVL C00141 BC00141 V=166.7
REFP 3 C00142 BC00142
CALL JOB:SEARCH-R1
SET P031 P006
SFTON P031
MOVL C00143 BC00143 V=166.7
SFTOF
MOVL C00144 BC00144 V=166.7
REFP 3 C00145 BC00145
CALL JOB:SEARCH-R1
SET P038 P006
SFTON P038
MOVL C00146 BC00146 V=166.7
REFP 3 C00147 BC00147
CALL JOB:SEARCH-R1
SET P038 P006
SFTON P038
MOVL C00148 BC00148 V=166.7
SFTOF
MOVL C00149 BC00149 V=166.7
REFP 3 C00150 BC00150
CALL JOB:SEARCH-R1
SET P039 P006
SFTON P039
MOVL C00151 BC00151 V=166.7
REFP 3 C00152 BC00152
CALL JOB:SEARCH-R1
SET P039 P006
SFTON P039
MOVL C00153 BC00153 V=166.7
MOVJ C00154 BC00154 VJ=100.00
SFTOF
MOVJ C00155 BC00155 VJ=100.00
MOVL C00156 BC00156 V=166.7
REFP 3 C00157 BC00157
CALL JOB:SEARCH-R1
SET P032 P006
SFTON P032
MOVL C00158 BC00158 V=166.7
REFP 3 C00159 BC00159
CALL JOB:SEARCH-R1
SET P032 P006
SFTON P032
MOVL C00160 BC00160 V=166.7
MOVL C00161 BC00161 V=166.7
SFTOF
MOVL C00162 BC00162 V=166.7
REFP 3 C00163 BC00163
CALL JOB:SEARCH-R1
SET P033 P006
SFTON P033
MOVL C00164 BC00164 V=166.7
REFP 3 C00165 BC00165
CALL JOB:SEARCH-R1
SET P033 P006
SFTON P033
MOVL C00166 BC00166 V=166.7
SFTOF
MOVL C00167 BC00167 V=166.7
REFP 3 C00168 BC00168
CALL JOB:SEARCH-R1
SET P040 P006
SFTON P040
MOVL C00169 BC00169 V=166.7
REFP 3 C00170 BC00170
CALL JOB:SEARCH-R1
SET P040 P006
SFTON P040
MOVL C00171 BC00171 V=166.7
MOVL C00172 BC00172 V=166.7
REFP 3 C00173 BC00173
CALL JOB:SEARCH-R1
SET P041 P006
SFTON P041
MOVL C00174 BC00174 V=166.7
REFP 3 C00175 BC00175
CALL JOB:SEARCH-R1
SET P041 P006
SFTON P041
MOVL C00176 BC00176 V=166.7
MOVL C00177 BC00177 V=333.3
'Path VIA1528
SFTOF
MOVL C00178 BC00178 V=166.7
REFP 3 C00179 BC00179
CALL JOB:SEARCH-R1
SET P034 P006
SFTON P034
MOVL C00180 BC00180 V=166.7
REFP 3 C00181 BC00181
CALL JOB:SEARCH-R1
SET P034 P006
SFTON P034
MOVL C00182 BC00182 V=166.7
MOVL C00183 BC00183 V=166.7
MOVJ C00184 BC00184 VJ=100.00
'Path S1527
SFTOF
MOVJ C00185 BC00185 VJ=40.00 PL=4 DEC=50
MOVJ C00186 BC00186 VJ=40.00 PL=4
MOVL C00187 BC00187 V=166.7
REFP 3 C00188 BC00188
CALL JOB:SEARCH-R1
SET P035 P006
SFTON P035
MOVL C00189 BC00189 V=166.7
REFP 3 C00190 BC00190
CALL JOB:SEARCH-R1
SET P035 P006
SFTON P035
MOVL C00191 BC00191 V=166.7
SFTOF
MOVL C00192 BC00192 V=250.0
REFP 3 C00193 BC00193
CALL JOB:SEARCH-R1
SET P036 P006
SFTON P036
MOVL C00194 BC00194 V=166.7
REFP 3 C00195 BC00195
CALL JOB:SEARCH-R1
SET P036 P006
SFTON P036
MOVL C00196 BC00196 V=166.7
MOVL C00197 BC00197 V=250.0
'Path W1520
SFTOF
REFP 3 C00198 BC00198
CALL JOB:SEARCH-R1
SET P037 P006
SFTON P037
MOVL C00199 BC00199 V=166.7
REFP 3 C00200 BC00200
CALL JOB:SEARCH-R1
SET P037 P006
SFTON P037
MOVL C00201 BC00201 V=166.7
SFTOF
MOVJ C00202 BC00202 VJ=40.00
MOVJ C00203 BC00203 VJ=100.00
PAUSE
'KONIEC SZUKANIA PRAWEGO BOCZKA
MOVJ C00204 BC00204 VJ=100.00
SFTON P035
MOVL C00205 BC00205 V=166.7 PL=0
REFP 1 C00206 BC00206
REFP 2 C00207 BC00207
MACRO1 MJ#(0) ARGF7
ARCON
SFTON P035
MOVL C00208 BC00208 V=12.5
ARCOF
MOVL C00209 BC00209 V=400.0
MOVL C00210 BC00210 V=1000.0
SFTOF
'Path W1521
SFTOF
SFTON P024
MOVJ C00211 BC00211 VJ=100.00
MOVJ C00212 BC00212 VJ=100.00
MOVJ C00213 BC00213 VJ=50.00
SFTON P034
MOVL C00214 BC00214 V=166.7 PL=0
REFP 1 C00215 BC00215
REFP 2 C00216 BC00216
MACRO1 MJ#(0) ARGF7
ARCON
SFTON P041
MOVL C00217 BC00217 V=11.7
SFTON P040
MOVL C00218 BC00218 V=11.7
SFTON P033
MOVL C00219 BC00219 V=11.7
MOVL C00220 BC00220 V=11.7
ARCOF
MOVL C00221 BC00221 V=166.7
SFTOF
'Path W1522
SFTOF
SFTON P036
MOVJ C00222 BC00222 VJ=100.00
MOVJ C00223 BC00223 VJ=100.00
MOVJ C00224 BC00224 VJ=100.00
MOVJ C00225 BC00225 VJ=100.00
SFTON P036
MOVL C00226 BC00226 V=166.7 PL=0
REFP 1 C00227 BC00227
REFP 2 C00228 BC00228
MACRO1 MJ#(0) ARGF9
ARCON
SFTON P037
MOVL C00229 BC00229 V=13.3
MOVL C00230 BC00230 V=13.3
MOVL C00231 BC00231 V=13.3
ARCOF
MOVL C00232 BC00232 V=166.7
MOVL C00233 BC00233 V=1000.0
SFTOF
'Path W1523
SFTOF
MOVJ C00234 BC00234 VJ=100.00
MOVJ C00235 BC00235 VJ=100.00
SFTOF
SFTON P031
MOVL C00236 BC00236 V=166.7 PL=0
REFP 1 C00237 BC00237
REFP 2 C00238 BC00238
MACRO1 MJ#(0) ARGF9
ARCON
MOVL C00239 BC00239 V=11.7
SFTON P038
MOVL C00240 BC00240 V=11.7
SFTON P039
MOVL C00241 BC00241 V=11.7
SFTON P032
MOVL C00242 BC00242 V=11.7
MOVL C00243 BC00243 V=11.7
ARCOF
MOVL C00244 BC00244 V=166.7
MOVL C00245 BC00245 V=1000.0
SFTOF
'Path W1524
SFTOF
SFTON P036
MOVJ C00246 BC00246 VJ=100.00
MOVJ C00247 BC00247 VJ=100.00
MOVJ C00248 BC00248 VJ=100.00
MOVL C00249 BC00249 V=166.7 PL=0
REFP 1 C00250 BC00250
REFP 2 C00251 BC00251
MACRO1 MJ#(0) ARGF9
ARCON
SFTON P035
MOVL C00252 BC00252 V=12.5
MOVL C00253 BC00253 V=12.5
MOVL C00254 BC00254 V=12.5
MOVL C00255 BC00255 V=12.5
MOVL C00256 BC00256 V=12.5
MOVL C00257 BC00257 V=12.5
ARCOF
MOVL C00258 BC00258 V=166.7
MOVL C00259 BC00259 V=1000.0
MOVJ C00260 BC00260 VJ=100.00
SFTOF
'Path W1531
SFTOF
MOVJ C00261 BC00261 VJ=100.00
SFTON P037
MOVJ C00262 BC00262 VJ=30.00
MOVL C00263 BC00263 V=166.7 PL=0
REFP 1 C00264 BC00264
REFP 2 C00265 BC00265
MACRO1 MJ#(0) ARGF9
ARCON
MOVL C00266 BC00266 V=10.3
MOVL C00267 BC00267 V=10.3
MOVL C00268 BC00268 V=10.3
SFTOF
SFTON P030
MOVL C00269 BC00269 V=11.7
MOVL C00270 BC00270 V=11.7
MOVL C00271 BC00271 V=11.7
MOVL C00272 BC00272 V=11.7
MOVL C00273 BC00273 V=11.7
MOVL C00274 BC00274 V=11.7
MOVL C00275 BC00275 V=11.7
MOVL C00276 BC00276 V=11.7
ARCOF
MOVL C00277 BC00277 V=166.7
SFTOF
MOVL C00278 BC00278 V=1000.0
MOVJ C00279 BC00279 VJ=100.00
MOVJ C00280 BC00280 VJ=100.00
CALL JOB:CLEAN-R1_LONG
MOVJ C00281 BC00281 VJ=100.00
MOVJ C00282 BC00282 VJ=100.00
'POCZATEK SZUKANIA LEWEGO BOCZKA
MOVJ C00283 BC00283 VJ=100.00
MOVL C00284 BC00284 V=166.7
REFP 3 C00285 BC00285
CALL JOB:SEARCH-R1
SET P021 P006
SFTON P021
MOVL C00286 BC00286 V=166.7
REFP 3 C00287 BC00287
CALL JOB:SEARCH-R1
SET P021 P006
SFTON P021
MOVL C00288 BC00288 V=166.7
SFTOF
'Path S1526
SFTOF
MOVL C00289 BC00289 V=166.7
MOVL C00290 BC00290 V=166.7
REFP 3 C00291 BC00291
CALL JOB:SEARCH-R1
SET P022 P006
SFTON P022
MOVL C00292 BC00292 V=166.7
REFP 3 C00293 BC00293
CALL JOB:SEARCH-R1
SET P022 P006
SFTON P022
MOVL C00294 BC00294 V=166.7
SFTOF
MOVL C00295 BC00295 V=166.7
REFP 3 C00296 BC00296
CALL JOB:SEARCH-R1
SET P042 P006
SFTON P042
MOVL C00297 BC00297 V=166.7
REFP 3 C00298 BC00298
CALL JOB:SEARCH-R1
SET P042 P006
SFTON P042
MOVL C00299 BC00299 V=166.7
SFTOF
MOVL C00300 BC00300 V=166.7
REFP 3 C00301 BC00301
CALL JOB:SEARCH-R1
SET P043 P006
SFTON P043
MOVL C00302 BC00302 V=166.7
REFP 3 C00303 BC00303
CALL JOB:SEARCH-R1
SET P043 P006
SFTON P043
MOVL C00304 BC00304 V=166.7
SFTOF
MOVL C00305 BC00305 V=166.7
REFP 3 C00306 BC00306
CALL JOB:SEARCH-R1
SET P023 P006
SFTON P023
MOVL C00307 BC00307 V=166.7
REFP 3 C00308 BC00308
CALL JOB:SEARCH-R1
SET P023 P006
SFTON P023
MOVL C00309 BC00309 V=166.7
MOVL C00310 BC00310 V=166.7
SFTOF
MOVL C00311 BC00311 V=166.7
REFP 3 C00312 BC00312
CALL JOB:SEARCH-R1
SET P024 P006
SFTON P024
MOVL C00313 BC00313 V=166.7
REFP 3 C00314 BC00314
CALL JOB:SEARCH-R1
SET P024 P006
SFTON P024
MOVL C00315 BC00315 V=166.7
MOVL C00316 BC00316 V=166.7
REFP 3 C00317 BC00317
CALL JOB:SEARCH-R1
SET P044 P006
SFTON P044
MOVL C00318 BC00318 V=166.7
REFP 3 C00319 BC00319
CALL JOB:SEARCH-R1
SET P044 P006
SFTON P044
MOVL C00320 BC00320 V=166.7
SFTOF
MOVL C00321 BC00321 V=166.7
REFP 3 C00322 BC00322
CALL JOB:SEARCH-R1
SET P045 P006
SFTON P045
MOVL C00323 BC00323 V=166.7
REFP 3 C00324 BC00324
CALL JOB:SEARCH-R1
SET P045 P006
SFTON P045
MOVL C00325 BC00325 V=166.7
MOVL C00326 BC00326 V=333.3
'Path VIA1528
SFTOF
MOVL C00327 BC00327 V=166.7
REFP 3 C00328 BC00328
CALL JOB:SEARCH-R1
SET P025 P006
SFTON P025
MOVL C00329 BC00329 V=166.7
REFP 3 C00330 BC00330
CALL JOB:SEARCH-R1
SET P025 P006
SFTON P025
MOVL C00331 BC00331 V=166.7
MOVL C00332 BC00332 V=166.7
'Path S1527
SFTOF
MOVL C00333 BC00333 V=166.7
REFP 3 C00334 BC00334
CALL JOB:SEARCH-R1
SET P026 P006
SFTON P026
MOVL C00335 BC00335 V=166.7
REFP 3 C00336 BC00336
CALL JOB:SEARCH-R1
SET P026 P006
SFTON P026
MOVL C00337 BC00337 V=166.7
SFTOF
MOVJ C00338 BC00338 VJ=100.00
MOVJ C00339 BC00339 VJ=100.00
MOVL C00340 BC00340 V=166.7
REFP 3 C00341 BC00341
CALL JOB:SEARCH-R1
SET P027 P006
SFTON P027
MOVL C00342 BC00342 V=166.7
REFP 3 C00343 BC00343
CALL JOB:SEARCH-R1
SET P027 P006
SFTON P027
MOVL C00344 BC00344 V=166.7
MOVJ C00345 BC00345 VJ=100.00
MOVJ C00346 BC00346 VJ=100.00
SFTOF
MOVL C00347 BC00347 V=166.7
'Path W1520
REFP 3 C00348 BC00348
CALL JOB:SEARCH-R1
SET P028 P006
SFTON P028
MOVL C00349 BC00349 V=166.7
REFP 3 C00350 BC00350
CALL JOB:SEARCH-R1
SET P028 P006
SFTON P028
MOVL C00351 BC00351 V=166.7
SFTOF
MOVJ C00352 BC00352 VJ=100.00
'START SPAWANIA LEWEGO BOCZKA
MOVJ C00353 BC00353 VJ=100.00
MACRO1 MJ#(0) ARGF7
SFTON P027
MOVL C00354 BC00354 V=166.7
ARCON
MOVL C00355 BC00355 V=12.5
ARCOF
SFTOF
MOVL C00356 BC00356 V=166.7
MOVJ C00357 BC00357 VJ=50.00
MACRO1 MJ#(0) ARGF7
MOVJ C00358 BC00358 VJ=80.00
SFTON P025
MOVL C00359 BC00359 V=166.7
ARCON
SFTON P045
MOVL C00360 BC00360 V=13.3
SFTON P044
MOVL C00361 BC00361 V=13.3
SFTON P024
MOVL C00362 BC00362 V=13.3
MOVL C00363 BC00363 V=13.3
ARCOF
MOVJ C00364 BC00364 VJ=20.00
SFTOF
MOVJ C00365 BC00365 VJ=100.00
MOVJ C00366 BC00366 VJ=80.00
MOVJ C00367 BC00367 VJ=100.00
SFTON P027
MOVL C00368 BC00368 V=166.7
ARCON
SFTON P028
MOVL C00369 BC00369 V=12.5
MOVL C00370 BC00370 V=12.5
ARCOF
SFTOF
MOVL C00371 BC00371 V=166.7
MOVJ C00372 BC00372 VJ=40.00
MOVJ C00373 BC00373 VJ=40.00
MOVJ C00374 BC00374 VJ=100.00
SFTON P022
MOVL C00375 BC00375 V=166.7
ARCON
SFTON P042
MOVL C00376 BC00376 V=13.3
SFTON P043
MOVL C00377 BC00377 V=13.3
SFTON P023
MOVL C00378 BC00378 V=13.3
MOVL C00379 BC00379 V=13.3
ARCOF
SFTOF
MOVL C00380 BC00380 V=166.7
MOVJ C00381 BC00381 VJ=100.00
MOVJ C00382 BC00382 VJ=100.00
SFTON P026
MOVL C00383 BC00383 V=166.7
ARCON
MOVL C00384 BC00384 V=13.3
MOVL C00385 BC00385 V=13.3
MOVL C00386 BC00386 V=13.3
MOVL C00387 BC00387 V=12.5
MOVL C00388 BC00388 V=12.5
MOVL C00389 BC00389 V=12.5
ARCOF
MOVL C00390 BC00390 V=166.7
SFTOF
MOVJ C00391 BC00391 VJ=100.00
MOVJ C00392 BC00392 VJ=100.00
MOVJ C00393 BC00393 VJ=100.00
SFTON P022
MOVL C00394 BC00394 V=166.7
ARCON
MOVL C00395 BC00395 V=10.0
MOVL C00396 BC00396 V=10.0
MOVL C00397 BC00397 V=10.0
MOVL C00398 BC00398 V=10.0
MOVL C00399 BC00399 V=11.7
MOVL C00400 BC00400 V=11.7
MOVL C00401 BC00401 V=11.7
MOVL C00402 BC00402 V=11.7
MOVL C00403 BC00403 V=11.7
MOVL C00404 BC00404 V=10.8
ARCOF
MOVL C00405 BC00405 V=166.7
MOVJ C00406 BC00406 VJ=100.00
SFTOF
MOVJ C00407 BC00407 VJ=100.00
MOVJ C00408 BC00408 VJ=100.00
MOVJ C00409 BC00409 VJ=100.00
END
